FUNCTION_BLOCK Test_TStreamAdd_Read_Short_STRING EXTENDS T_UnitTestBase
VAR
    Stream     : T_Stream(StreamLength := 2);
    ArgType    : E_ArgTypeId := E_ArgTypeId.Type_STRING;
    TestString : STRING(10)  := '0123456789';
END_VAR

METHOD  Init
VAR_INPUT
END_VAR
END_METHOD

{attribute 'analysis' := '-33'} // inhibit unused variable warning
METHOD RunTest

Stream.Init(2);

// add a STRING...
Stream.SetNextArgTypeId(ArgType);
Stream.Add_STRING(TestString);

Stream.SetReadPosition(0);

// check next arg type is correct...
AssertEquals_INT(Expected     := ArgType,
                           Actual       := Stream.GetNextArgTypeId(),
                           Message := 'Stream.GetNextArgTypeId()');

// check next value...	
AssertEquals_STRING(Expected     := TestString,
                              Actual       := Stream.Read_STRING(),
                              Message := 'Stream.Read_STRING()');

// check we are at the end of the stream..							
AssertEquals_UDINT(Expected     := Stream.StreamLength,
                             Actual       := Stream.ReadPosition,
                             Message := 'Stream.ReadPosition');

TestCompleted := TRUE;
END_METHOD

END_FUNCTION_BLOCK

(* stored: Version 1.1.0.1, ProductVersion 3.1.4024.12
   POU Test_TStreamAdd_Read_Short_STRING: Id {26a7714d-6abb-4cdf-ba46-ea1540b1ab15}, SpecialFunc None
   Method Init: Id {38735707-e61a-4d1d-8768-e26d2b536584}
   Method RunTest: Id {9ab42624-80c5-476c-9f84-7c8f0aa94f4e} *)
